TYPE ST_SpindleParameters :
STRUCT
    
// Invertek Optidrive E3 Modbus Register Mapping Parameters

    
nMaxSpeedLimit		: UINT; //Modbus RTU Register 129
nMinSpeedLimit	    : UINT; //Modbus RTU Register 130
nAccelRampTime		: UINT; //Modbus RTU Register 131
nDecelRampTime		: UINT; //Modbus RTU Register 132
nStopMode			: UINT; //Modbus RTU Register 133
nMotorRatedVoltage	: UINT; //Modbus RTU Register 135
nMotorRatedCurrent  : UINT; //Modbus RTU Register 136
nMotorRatedFrequency: UINT; //Modbus RTU Register 137
nMotorRatedSpeed    : UINT; //Modbus RTU Register 138
nApplicationMode    : UINT; //Modbus RTU Register 141
nRelayOutputFunction: UINT; //Modbus RTU Register 146
nUserPGain          : UINT; //Modbus RTU Register 169
nUserIConstant      : UINT; //Modbus RTU Register 170
nMotorControlMode   : UINT; //Modbus RTU Register 179
nMaximumCurrentLimit: UINT; //Modbus RTU Register 182



END_STRUCT
END_TYPE

(* stored: Version 1.1.0.1, ProductVersion 3.1.4024.9
   DUT ST_SpindleParameters: Id {904f6f5b-ce80-4d8c-a494-929ac264aba0} *)
